INTERFACE I_RpcHandler

METHOD Handle
VAR_INPUT
	Parameters : I_RpcParameters;
	Response : I_SynchronousRpcResponse;
END_VAR
END_METHOD

END_INTERFACE

(* stored: Version 1.1.0.1, ProductVersion 3.1.4024.12
   Itf I_RpcHandler: Id {443f7afb-60e8-4caf-9dc0-bacc792c6826}
   Method Handle: Id {4ab0dfeb-bf05-4348-9808-69f446eb5d69} *)
